FUNCTION_BLOCK FB_EdgeDetector
VAR_INPUT
	inputValue : BOOL;
	DoublePressedTime: UINT;
END_VAR
VAR_OUTPUT
	risingEdge : BOOL;
	fallingEdge : BOOL;
	DoublePressed: BOOL;
END_VAR
VAR
	inputValue_old : BOOL;
	OncePressed: BOOL := FALSE;
	DoublePressedcounter: UINT := 0;
END_VAR

risingEdge := FALSE;
fallingEdge := FALSE;
DoublePressed := FALSE;

IF inputValue <> inputValue_old THEN
	IF inputValue = TRUE THEN
		risingEdge := TRUE;
		IF OncePressed = FALSE THEN
			OncePressed := TRUE;
		ELSE
			OncePressed := FALSE;
			DoublePressed := TRUE;
			DoublePressedcounter := 0;
		END_IF
	ELSE
		fallingEdge := TRUE;
	END_IF
END_IF
inputValue_old := inputValue;
IF OncePressed = TRUE THEN
	IF DoublePressedcounter >= DoublePressedTime THEN
		OncePressed := FALSE;
		DoublePressedcounter := 0;
	ELSE
		DoublePressedcounter := DoublePressedcounter + 1;
	END_IF	
END_IF

END_FUNCTION_BLOCK

(* stored: Version 1.1.0.1, ProductVersion 3.1.4024.13
   POU FB_EdgeDetector: Id {b5174619-237e-4dd2-8278-f66c17ef7d36}, SpecialFunc None *)
